FUNCTION CharIsNumber : BOOL
VAR_INPUT
   bChar : BYTE; // char to check
END_VAR

// check bChar is in numbr range of ascii
CharIsNumber := (bChar >= 48 AND bChar <= 57);

END_FUNCTION

(* stored: Version 1.1.0.1, ProductVersion 3.1.4024.9
   POU CharIsNumber: Id {d8360be8-ce72-4bcc-bb95-e4c62b585976}, SpecialFunc None *)
